VAR_GLOBAL
    EnableAdsLogger : BOOL := TRUE;
    EnableTcEventLogging : BOOL := FALSE;
    TraceLevel : TcEventSeverityExt := TcEventSeverityExt.Verbose;
	Trace : Trace<10> := (TraceLevel := TraceLevel);
	TcEventLogger : TcEventLogger(Trace);
	AdsLogger : AdsLogger(Trace);
END_VAR

(* stored: Version 1.1.0.1, ProductVersion 3.1.4026.18
   GVL GvlTrace: Id {a08d82f5-c40f-43ad-8071-187f0f8bb6e7} *)
